Omron CX-Programmer project NewProject (CX-Programmer 9.80)

# PLC NewPLC1: CQM1H CPU51

## Global symbols (name address type ; comment)
0.06 BOOL  ; CAP ZERO ELEV BRAS
0.07 BOOL  ; F-C H ELEV BRAS(active_low)
0.08 BOOL  ; ranger complet
0.09 BOOL  ; F-C H ELEV ROUL
0.11 BOOL  ; F-C SEC ELEV BRAS
0.12 BOOL  ; F-C TIRANT BRAS
100.00 BOOL  ; MONT ELEV BRAS
100.01 BOOL  ; DESCENT ELEV BRAS
100.02 BOOL  ; MONT ELEV ROUL
100.03 BOOL  ; DESCENT ELEV ROUL
100.06 BOOL  ; M-ROUL FIXE
100.10 BOOL  ; VITESSE1 ELEV BRAS
100.11 BOOL  ; VITESSE2 ELEV BRAS
100.13 BOOL  ; VITESSE1 ELEV ROUL
101.00 BOOL  ; VITESSE3 ROUL FIXE
101.08 BOOL  ; FREIN ELEV BRAS
101.09 BOOL  ; FREIN ELEV ROUL
101.10 BOOL  ; INSER COMMANDE
101.11 BOOL  ; SIRENE
101.13 BOOL  ; M-COUROIE ENTREE
102.00 BOOL  ; M-ELEV BRAS
102.01 BOOL  ; M-ROUL BOX
102.02 BOOL  ; OUVER BRAS
102.03 BOOL  ; FERME BRAS
102.06 BOOL  ; SOULEV COURROIE
102.08 BOOL  ; M/D CENTREUR
102.09 BOOL  ; AVANT CHAINE
102.10 BOOL  ; ARRIERE CHAINE
102.11 BOOL  ; VITESSE1 CHAINE
102.12 BOOL  ; PASSARELLA  AVANT
102.14 BOOL  ; PASSARELLA  ARRIERE
102.15 BOOL  ; PASSARELLA  ARRIERE Vitesse 1
116.00 BOOL  ; presence box avec obligation du centrerur ou non box
116.01 BOOL  ; front montant cateur zero elev bras
116.10 BOOL  ; automatique chaine
116.11 BOOL  ; man/auto
117.06 BOOL  ; condition securiter elev rolo en position bas
118.10 BOOL  ; position acutuelle>position de reference
118.11 BOOL  ; position_actuelle<positioin_de_reference
119.14 BOOL  ; button_zero
120.00 BOOL  ; button_zero
120.01 BOOL  ; button_start_cycle_automatique
121.00 BOOL  ; UP_cent_hmi_button
121.01 BOOL  ; descent_centrure_hmi_button
121.02 BOOL  ; BUTTON_chaine_avant_hmi
121.03 BOOL  ; button_chaine_arriere_hmi
140.00 BOOL  ; front mont hr1.00
170.00 BOOL  ; condition monter et frein elev bras
170.01 BOOL  ; condition descente elev bras
1.00 BOOL  ; CAP BRAS OUVERT
1.01 BOOL  ; CAP BRAS FERMEE
1.02 BOOL  ; PH-C DEBORD BOX
1.03 BOOL  ; cap alignement elev rolo et elev bra
1.05 BOOL  ; capteur alignement table fixe et elev rolo
1.06 BOOL  ; CAP COURROIE BAS
1.07 BOOL  ; PH-C FILA CMPL
1.08 BOOL  ; PH-C DEBUT ROUL
1.09 BOOL  ; PH-C STOP FILA
1.10 BOOL  ; PH-C ROUL BOX
1.11 BOOL  ; PH-C P.A.P
1.14 BOOL  ; CENTREUR H
1.15 BOOL  ; CENTREUR BAS
2.00 BOOL  ; COMMANDE INSEREE
2.01 BOOL  ; DCL THERMIQUE
2.02 BOOL  ; ALARME INV
2.04 BOOL  ; switcheur_passarella_arriere
2.05 BOOL  ; switcheur_passarella_avant
2.06 BOOL  ; F-C BOX MACHINE
2.08 BOOL  ; F-C CHAINE AVANT
2.09 BOOL  ; FC_CHAINE_ARRIERE
2.10 BOOL  ; retour_partielle
2.12 BOOL  ; fc_zone_a_passarella
2.13 BOOL  ; passarella_en_avant
2.14 BOOL  ; PASSARELLA_en_arriere
2.15 BOOL  ; fc_zone_b_passarella
70.02 BOOL  ; condition monter elev rolo
70.03 BOOL  ; condition desencete elev rolo
71.03 BOOL  ; COND_Passarella_avnat
71.04 BOOL  ; cond_passarella_arriere
72.06 BOOL  ; condition_centrure
72.08 BOOL  ; condition_centrure
72.09 BOOL  ; condition_chaine_avant
72.10 BOOL  ; condition_chaine_arriere
HR0.00 BOOL  ; start-chargement-box-automatique
HR10.02 BOOL  ; condition pour descent au capteur zero (aligne au box )
HR10.03 BOOL  ; elev bras en  pos 0
HR10.13 BOOL  ; condition 0 elev rouleau
HR10.15 BOOL  ; machine en pos zero
HR11.00 BOOL  ; condition pour start cycle automatique
HR11.01 BOOL  ; condition pour depart du cycle_automatique
HR11.02 BOOL  ; machine en pos initiale avec alignement entre bras et rolo
HR11.03 BOOL  ; condition pour fin du cycle
HR13.00 BOOL  ; chercher table fixe vers l'haut
HR13.01 BOOL  ; chercher table fixe vers le bas
HR13.02 BOOL  ; table mobile  aligne au table fixe
HR13.03 BOOL  ; range complet table fix
HR1.00 BOOL  ; condition pour  elev bra en position exacte et bras fermer
HR1.05 BOOL  ; BT_complet_charging_box
HR2.01 BOOL  ; condition de chercher du elev rolo vers le haut
HR2.02 BOOL  ; condition de chercher du elev bras vers le bas
HR2.03 BOOL  ; condition monter elev rolo en fin du cycle
HR2.04 BOOL  ; condition chercher table fixe  vers le bas
HR2.05 BOOL  ; condition du chercher du table fixe vers le haut
HR3.00 BOOL  ; chaine en automatique
HR3.01 BOOL  ; centrure bas_automatique et manuelle
HR3.02 BOOL  ; etat_box_ready_to_go_out
HR3.03 BOOL  ; etat_BOX_out
HR3.04 BOOL  ; WAIT FOR EMPTY BOX
HR3.05 BOOL  ; BOX IS READY TO ENTER
HR3.06 BOOL  ; condition d'activation cent h man et auto
HR5.04 BOOL  ; Condition alarme generale
HR5.05 BOOL  ; ALARM CENTRURE
HR8.01 BOOL  ; ETAT ARRIERE PASSARELLA

## Program NewProgram1 (no task)

### Section Section1

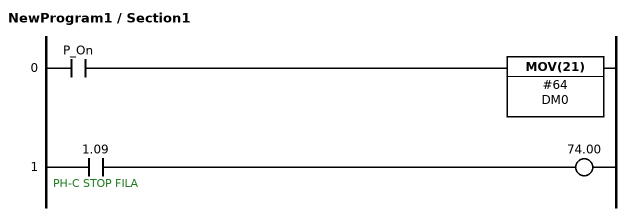
; rung 0
LD P_On
MOV(21) #64 DM0
; rung 1
LD 1.09  ; PH-C STOP FILA
OUT 74.00

### Section Section2

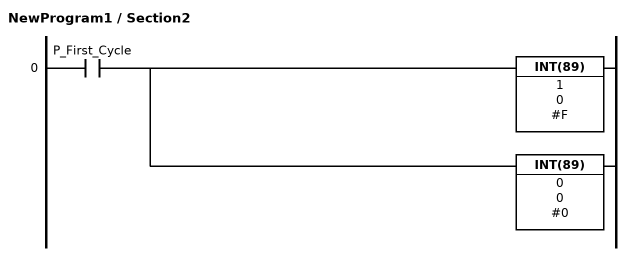
; rung 0
LD P_First_Cycle
INT(89) 1 0 #F
INT(89) 0 0 #0

### Section Section3

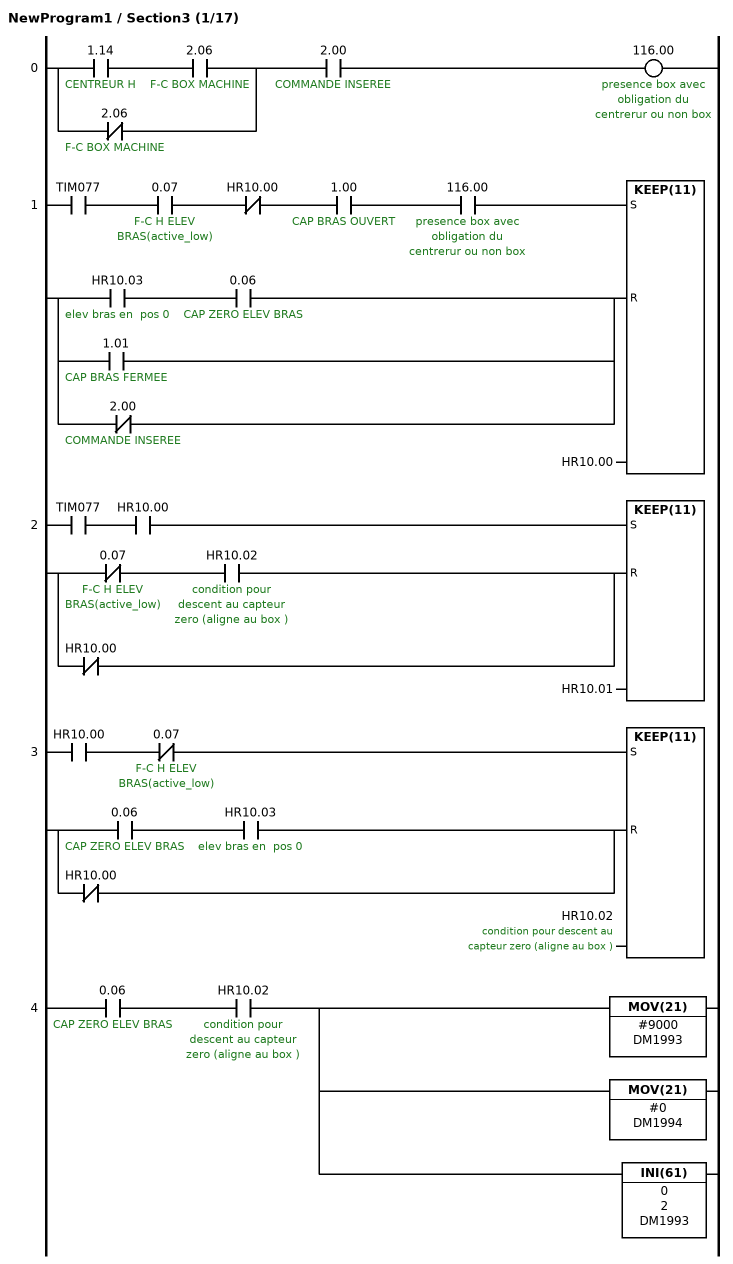
; rung 0
LD 1.14  ; CENTREUR H
AND 2.06  ; F-C BOX MACHINE
ORNOT 2.06  ; F-C BOX MACHINE
AND 2.00  ; COMMANDE INSEREE
OUT 116.00  ; presence box avec obligation du centrerur ou non box
; rung 1
LD TIM077
AND 0.07  ; F-C H ELEV BRAS(active_low)
ANDNOT HR10.00
AND 1.00  ; CAP BRAS OUVERT
AND 116.00  ; presence box avec obligation du centrerur ou non box
LD HR10.03  ; elev bras en  pos 0
AND 0.06  ; CAP ZERO ELEV BRAS
OR 1.01  ; CAP BRAS FERMEE
ORNOT 2.00  ; COMMANDE INSEREE
KEEP(11) HR10.00
; rung 2
LD TIM077
AND HR10.00
LDNOT 0.07  ; F-C H ELEV BRAS(active_low)
AND HR10.02  ; condition pour descent au capteur zero (aligne au box )
ORNOT HR10.00
KEEP(11) HR10.01
; rung 3
LD HR10.00
ANDNOT 0.07  ; F-C H ELEV BRAS(active_low)
LD 0.06  ; CAP ZERO ELEV BRAS
AND HR10.03  ; elev bras en  pos 0
ORNOT HR10.00
KEEP(11) HR10.02  ; condition pour descent au capteur zero (aligne au box )
; rung 4
LD 0.06  ; CAP ZERO ELEV BRAS
AND HR10.02  ; condition pour descent au capteur zero (aligne au box )
MOV(21) #9000 DM1993
MOV(21) #0 DM1994
INI(61) 0 2 DM1993

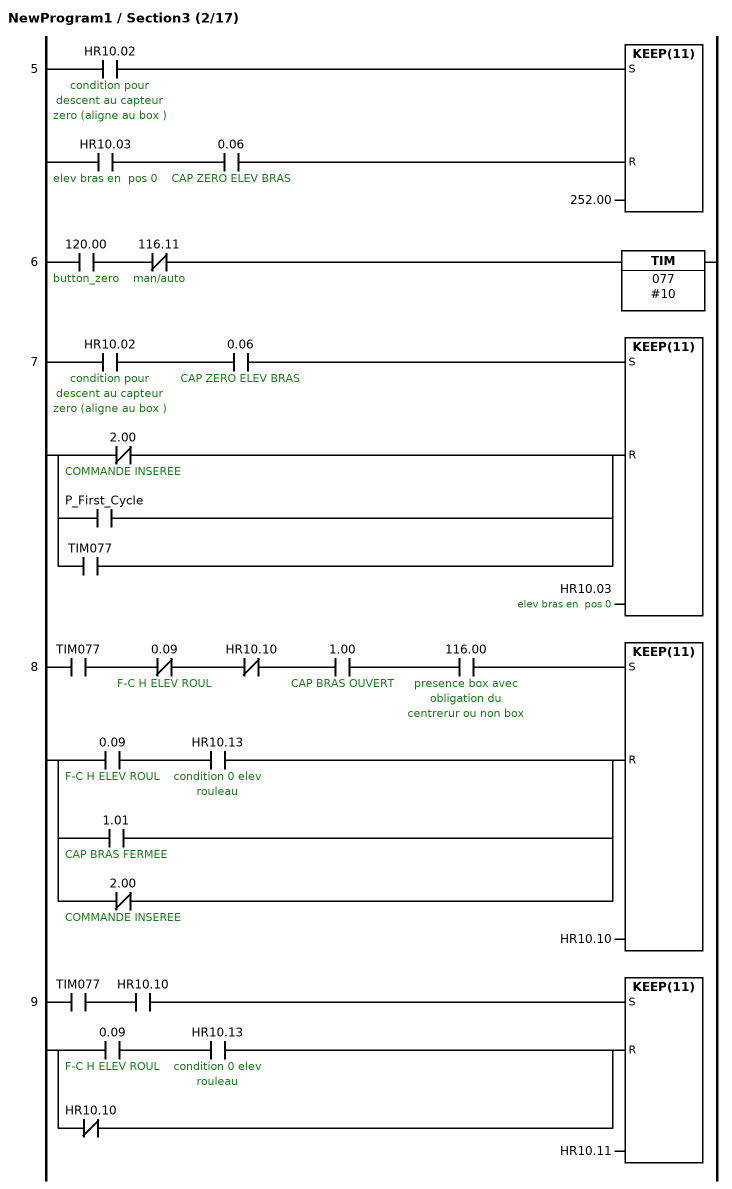
; rung 5
LD HR10.02  ; condition pour descent au capteur zero (aligne au box )
LD HR10.03  ; elev bras en  pos 0
AND 0.06  ; CAP ZERO ELEV BRAS
KEEP(11) 252.00
; rung 6
LD 120.00  ; button_zero
ANDNOT 116.11  ; man/auto
TIM 077 #10
; rung 7
LD HR10.02  ; condition pour descent au capteur zero (aligne au box )
AND 0.06  ; CAP ZERO ELEV BRAS
LDNOT 2.00  ; COMMANDE INSEREE
OR P_First_Cycle
OR TIM077
KEEP(11) HR10.03  ; elev bras en  pos 0
; rung 8
LD TIM077
ANDNOT 0.09  ; F-C H ELEV ROUL
ANDNOT HR10.10
AND 1.00  ; CAP BRAS OUVERT
AND 116.00  ; presence box avec obligation du centrerur ou non box
LD 0.09  ; F-C H ELEV ROUL
AND HR10.13  ; condition 0 elev rouleau
OR 1.01  ; CAP BRAS FERMEE
ORNOT 2.00  ; COMMANDE INSEREE
KEEP(11) HR10.10
; rung 9
LD TIM077
AND HR10.10
LD 0.09  ; F-C H ELEV ROUL
AND HR10.13  ; condition 0 elev rouleau
ORNOT HR10.10
KEEP(11) HR10.11

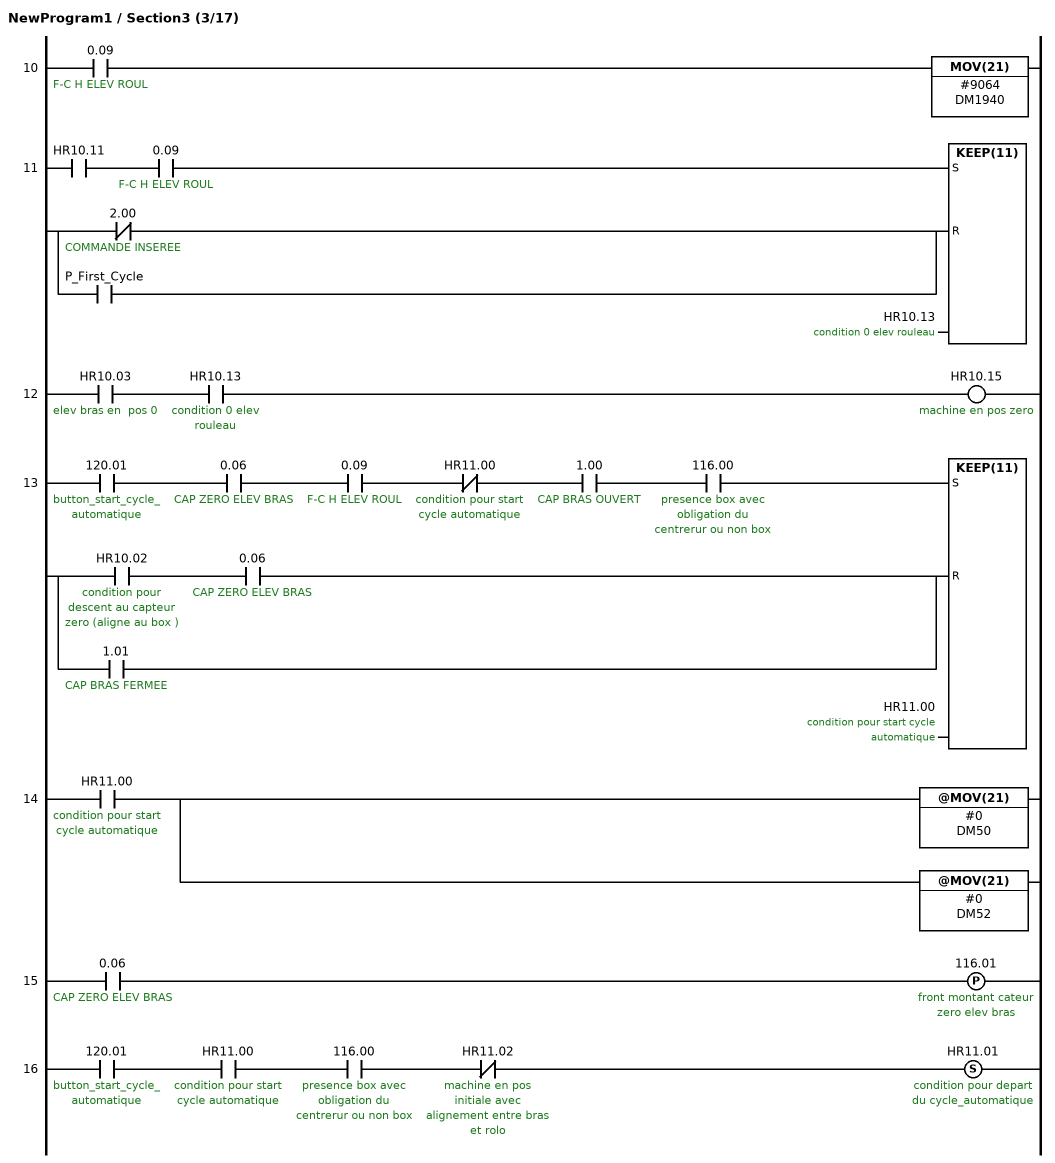
; rung 10
LD 0.09  ; F-C H ELEV ROUL
MOV(21) #9064 DM1940
; rung 11
LD HR10.11
AND 0.09  ; F-C H ELEV ROUL
LDNOT 2.00  ; COMMANDE INSEREE
OR P_First_Cycle
KEEP(11) HR10.13  ; condition 0 elev rouleau
; rung 12
LD HR10.03  ; elev bras en  pos 0
AND HR10.13  ; condition 0 elev rouleau
OUT HR10.15  ; machine en pos zero
; rung 13
LD 120.01  ; button_start_cycle_automatique
AND 0.06  ; CAP ZERO ELEV BRAS
AND 0.09  ; F-C H ELEV ROUL
ANDNOT HR11.00  ; condition pour start cycle automatique
AND 1.00  ; CAP BRAS OUVERT
AND 116.00  ; presence box avec obligation du centrerur ou non box
LD HR10.02  ; condition pour descent au capteur zero (aligne au box )
AND 0.06  ; CAP ZERO ELEV BRAS
OR 1.01  ; CAP BRAS FERMEE
KEEP(11) HR11.00  ; condition pour start cycle automatique
; rung 14
LD HR11.00  ; condition pour start cycle automatique
@MOV(21) #0 DM50
@MOV(21) #0 DM52
; rung 15
LD 0.06  ; CAP ZERO ELEV BRAS
DIFU(13) 116.01  ; front montant cateur zero elev bras
; rung 16
LD 120.01  ; button_start_cycle_automatique
AND HR11.00  ; condition pour start cycle automatique
AND 116.00  ; presence box avec obligation du centrerur ou non box
ANDNOT HR11.02  ; machine en pos initiale avec alignement entre bras et rolo
SET HR11.01  ; condition pour depart du cycle_automatique

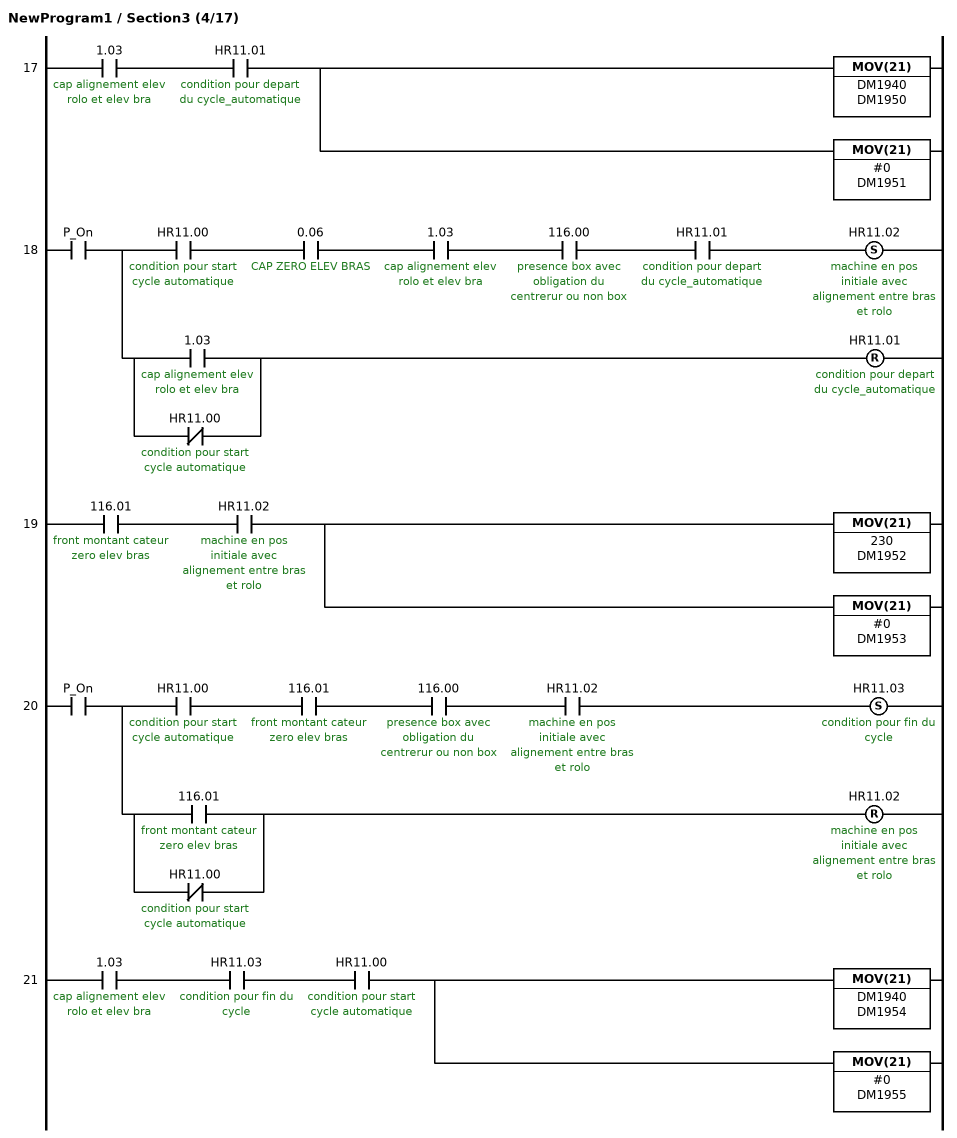
; rung 17
LD 1.03  ; cap alignement elev rolo et elev bra
AND HR11.01  ; condition pour depart du cycle_automatique
MOV(21) DM1940 DM1950
MOV(21) #0 DM1951
; rung 18
LD P_On
OUT TR0
AND HR11.00  ; condition pour start cycle automatique
AND 0.06  ; CAP ZERO ELEV BRAS
AND 1.03  ; cap alignement elev rolo et elev bra
AND 116.00  ; presence box avec obligation du centrerur ou non box
AND HR11.01  ; condition pour depart du cycle_automatique
SET HR11.02  ; machine en pos initiale avec alignement entre bras et rolo
LD TR0
LD 1.03  ; cap alignement elev rolo et elev bra
ORNOT HR11.00  ; condition pour start cycle automatique
ANDLD
RSET HR11.01  ; condition pour depart du cycle_automatique
; rung 19
LD 116.01  ; front montant cateur zero elev bras
AND HR11.02  ; machine en pos initiale avec alignement entre bras et rolo
MOV(21) 230 DM1952
MOV(21) #0 DM1953
; rung 20
LD P_On
OUT TR0
AND HR11.00  ; condition pour start cycle automatique
AND 116.01  ; front montant cateur zero elev bras
AND 116.00  ; presence box avec obligation du centrerur ou non box
AND HR11.02  ; machine en pos initiale avec alignement entre bras et rolo
SET HR11.03  ; condition pour fin du cycle
LD TR0
LD 116.01  ; front montant cateur zero elev bras
ORNOT HR11.00  ; condition pour start cycle automatique
ANDLD
RSET HR11.02  ; machine en pos initiale avec alignement entre bras et rolo
; rung 21
LD 1.03  ; cap alignement elev rolo et elev bra
AND HR11.03  ; condition pour fin du cycle
AND HR11.00  ; condition pour start cycle automatique
MOV(21) DM1940 DM1954
MOV(21) #0 DM1955

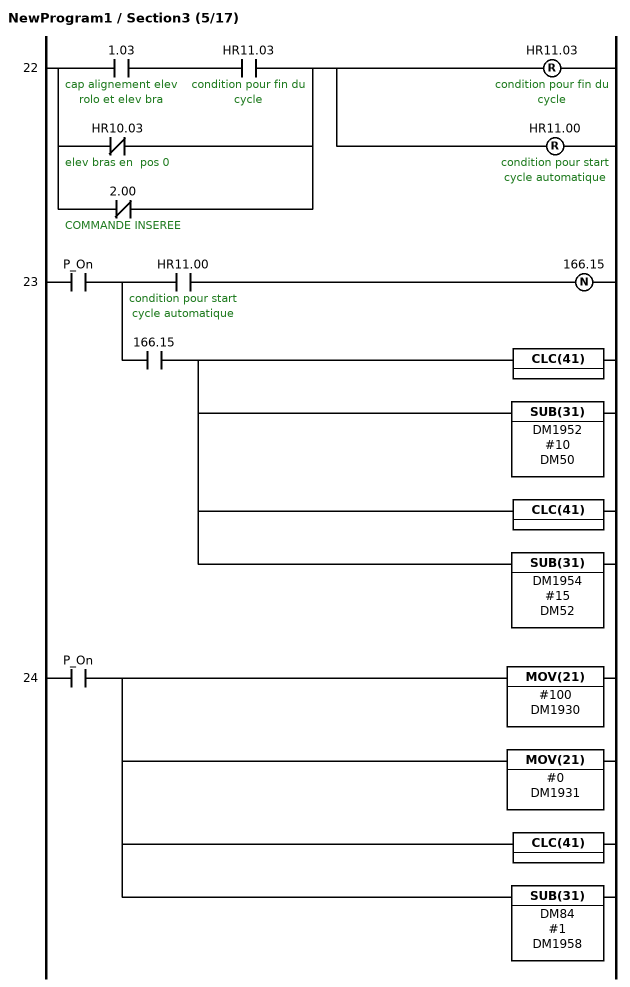
; rung 22
LD 1.03  ; cap alignement elev rolo et elev bra
AND HR11.03  ; condition pour fin du cycle
ORNOT HR10.03  ; elev bras en  pos 0
ORNOT 2.00  ; COMMANDE INSEREE
RSET HR11.03  ; condition pour fin du cycle
RSET HR11.00  ; condition pour start cycle automatique
; rung 23
LD P_On
OUT TR0
AND HR11.00  ; condition pour start cycle automatique
DIFD(14) 166.15
LD TR0
AND 166.15
CLC(41)
SUB(31) DM1952 #10 DM50
CLC(41)
SUB(31) DM1954 #15 DM52
; rung 24
LD P_On
MOV(21) #100 DM1930
MOV(21) #0 DM1931
CLC(41)
SUB(31) DM84 #1 DM1958

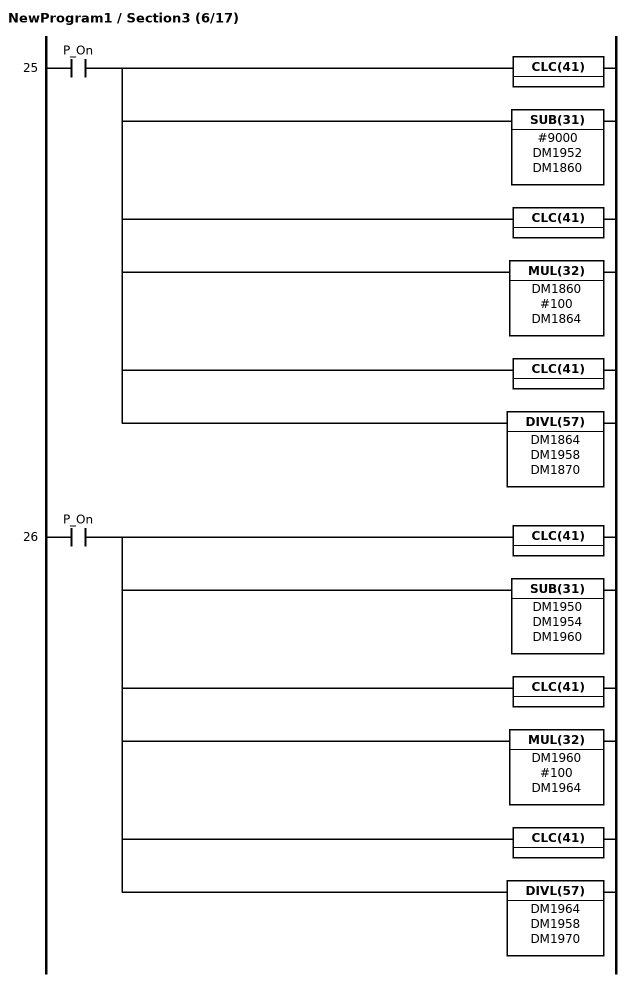
; rung 25
LD P_On
CLC(41)
SUB(31) #9000 DM1952 DM1860
CLC(41)
MUL(32) DM1860 #100 DM1864
CLC(41)
DIVL(57) DM1864 DM1958 DM1870
; rung 26
LD P_On
CLC(41)
SUB(31) DM1950 DM1954 DM1960
CLC(41)
MUL(32) DM1960 #100 DM1964
CLC(41)
DIVL(57) DM1964 DM1958 DM1970

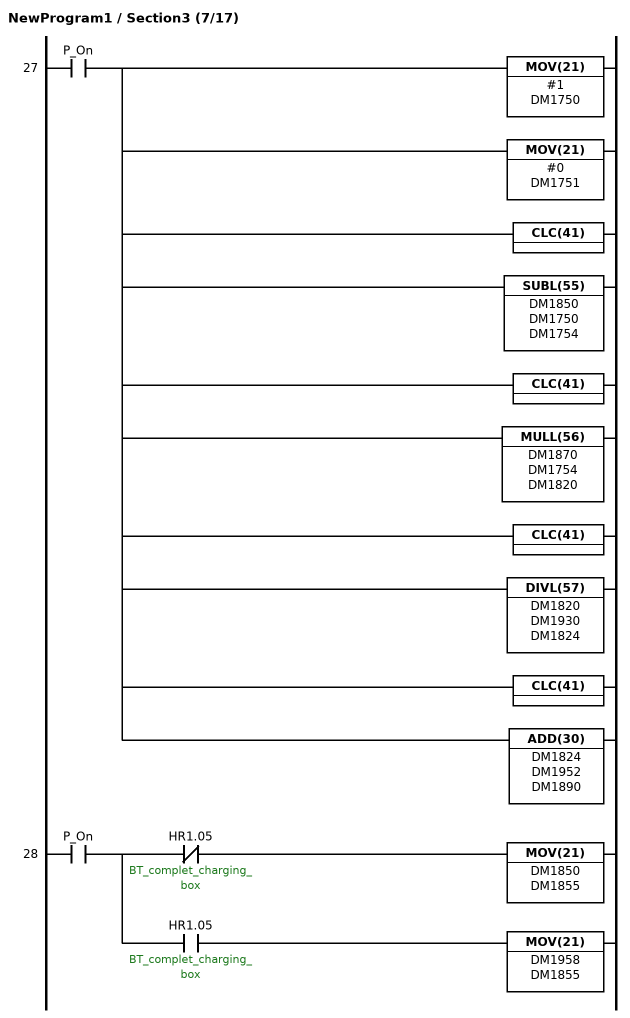
; rung 27
LD P_On
MOV(21) #1 DM1750
MOV(21) #0 DM1751
CLC(41)
SUBL(55) DM1850 DM1750 DM1754
CLC(41)
MULL(56) DM1870 DM1754 DM1820
CLC(41)
DIVL(57) DM1820 DM1930 DM1824
CLC(41)
ADD(30) DM1824 DM1952 DM1890
; rung 28
LD P_On
OUT TR0
ANDNOT HR1.05  ; BT_complet_charging_box
MOV(21) DM1850 DM1855
LD TR0
AND HR1.05  ; BT_complet_charging_box
MOV(21) DM1958 DM1855

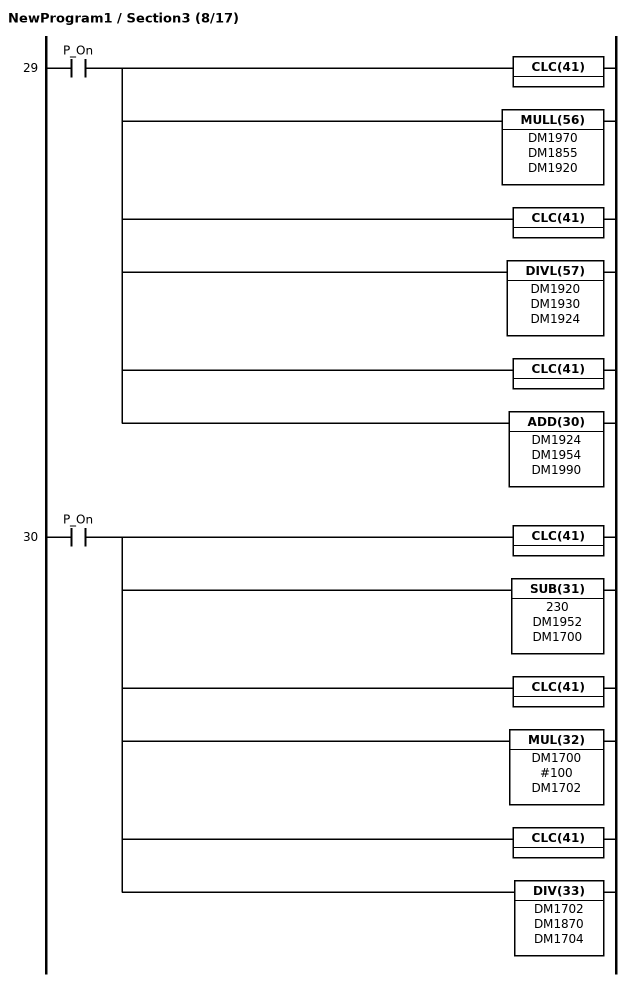
; rung 29
LD P_On
CLC(41)
MULL(56) DM1970 DM1855 DM1920
CLC(41)
DIVL(57) DM1920 DM1930 DM1924
CLC(41)
ADD(30) DM1924 DM1954 DM1990
; rung 30
LD P_On
CLC(41)
SUB(31) 230 DM1952 DM1700
CLC(41)
MUL(32) DM1700 #100 DM1702
CLC(41)
DIV(33) DM1702 DM1870 DM1704

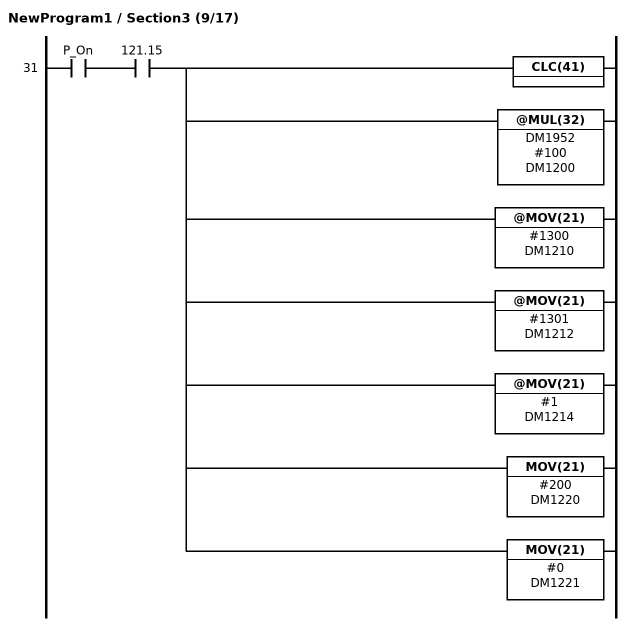
; rung 31
LD P_On
AND 121.15
CLC(41)
@MUL(32) DM1952 #100 DM1200
@MOV(21) #1300 DM1210
@MOV(21) #1301 DM1212
@MOV(21) #1 DM1214
MOV(21) #200 DM1220
MOV(21) #0 DM1221

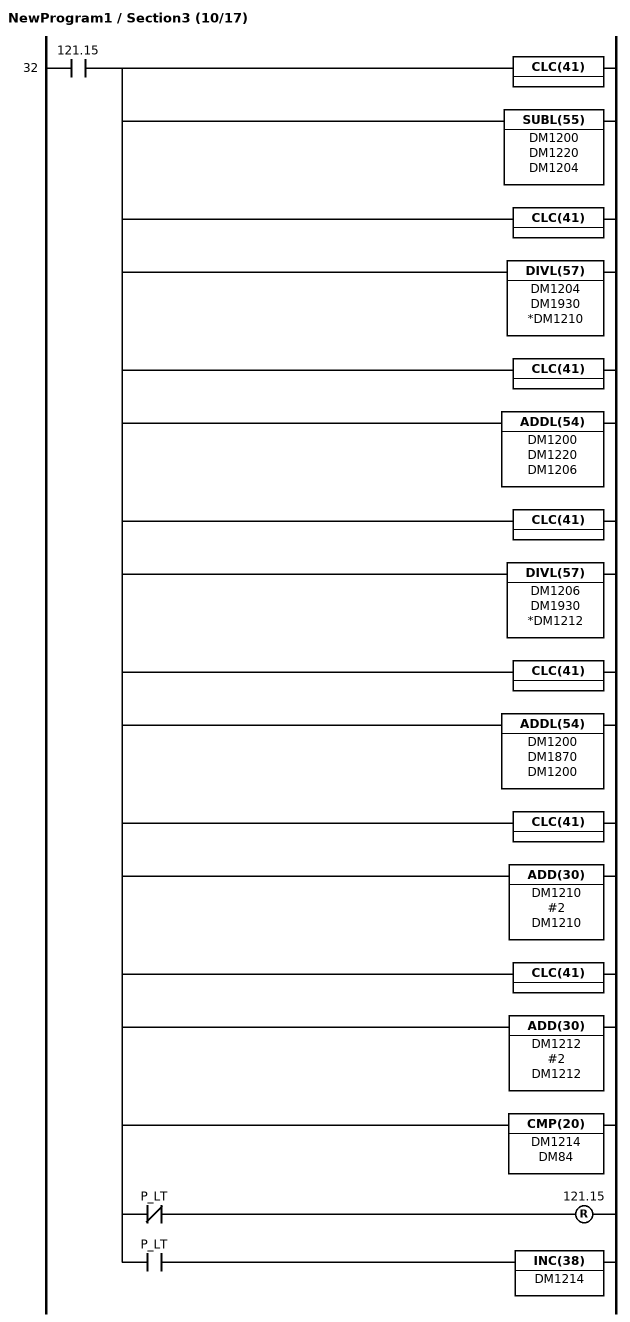
; rung 32
LD 121.15
OUT TR0
CLC(41)
SUBL(55) DM1200 DM1220 DM1204
CLC(41)
DIVL(57) DM1204 DM1930 *DM1210
CLC(41)
ADDL(54) DM1200 DM1220 DM1206
CLC(41)
DIVL(57) DM1206 DM1930 *DM1212
CLC(41)
ADDL(54) DM1200 DM1870 DM1200
CLC(41)
ADD(30) DM1210 #2 DM1210
CLC(41)
ADD(30) DM1212 #2 DM1212
CMP(20) DM1214 DM84
ANDNOT P_LT
RSET 121.15
LD TR0
AND P_LT
INC(38) DM1214

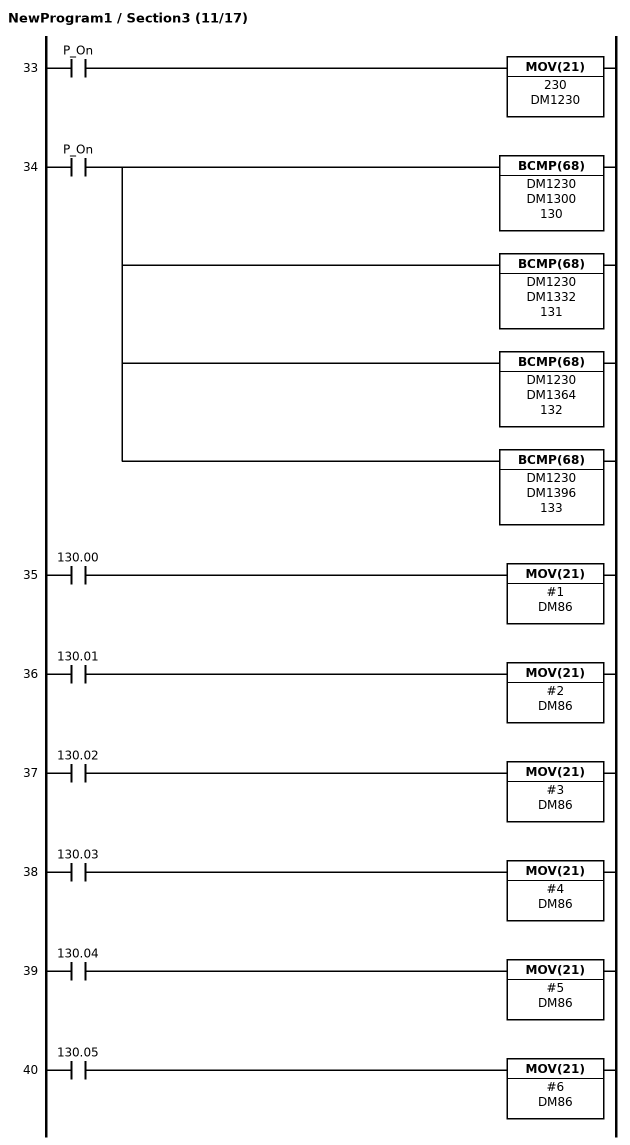
; rung 33
LD P_On
MOV(21) 230 DM1230
; rung 34
LD P_On
BCMP(68) DM1230 DM1300 130
BCMP(68) DM1230 DM1332 131
BCMP(68) DM1230 DM1364 132
BCMP(68) DM1230 DM1396 133
; rung 35
LD 130.00
MOV(21) #1 DM86
; rung 36
LD 130.01
MOV(21) #2 DM86
; rung 37
LD 130.02
MOV(21) #3 DM86
; rung 38
LD 130.03
MOV(21) #4 DM86
; rung 39
LD 130.04
MOV(21) #5 DM86
; rung 40
LD 130.05
MOV(21) #6 DM86

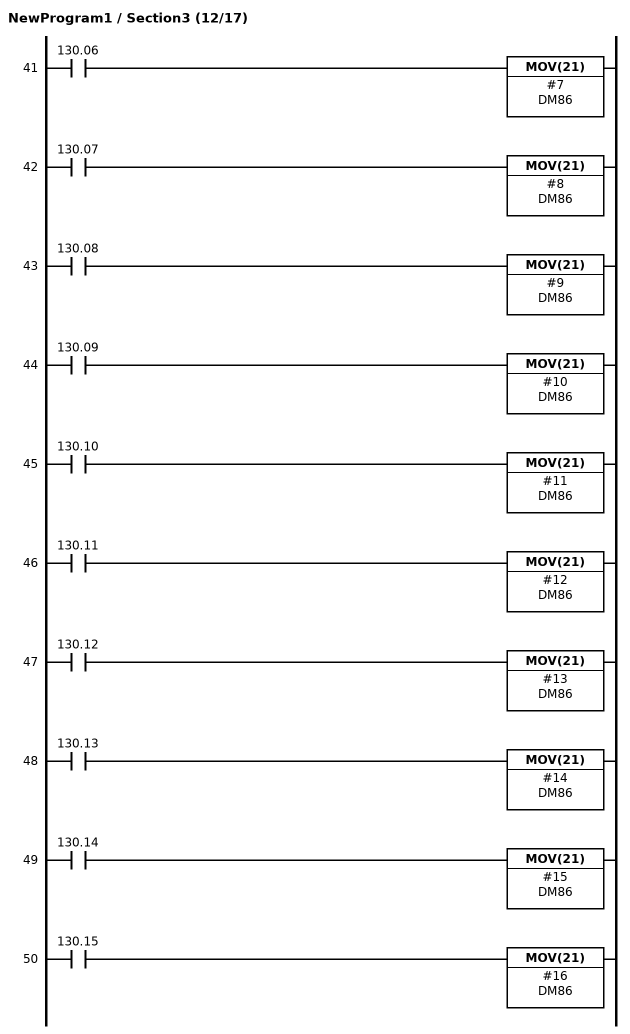
; rung 41
LD 130.06
MOV(21) #7 DM86
; rung 42
LD 130.07
MOV(21) #8 DM86
; rung 43
LD 130.08
MOV(21) #9 DM86
; rung 44
LD 130.09
MOV(21) #10 DM86
; rung 45
LD 130.10
MOV(21) #11 DM86
; rung 46
LD 130.11
MOV(21) #12 DM86
; rung 47
LD 130.12
MOV(21) #13 DM86
; rung 48
LD 130.13
MOV(21) #14 DM86
; rung 49
LD 130.14
MOV(21) #15 DM86
; rung 50
LD 130.15
MOV(21) #16 DM86

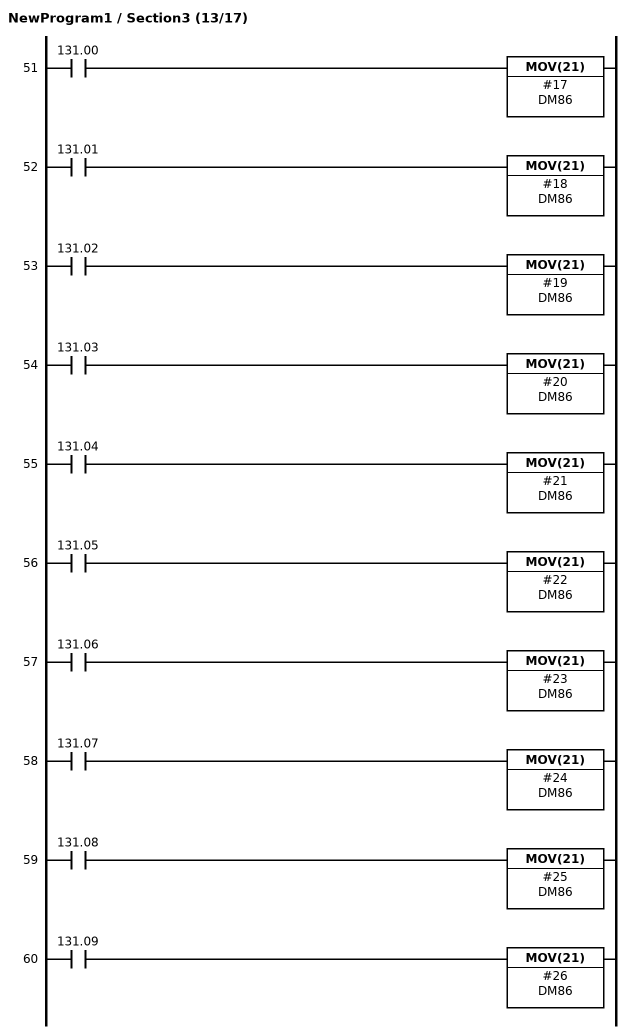
; rung 51
LD 131.00
MOV(21) #17 DM86
; rung 52
LD 131.01
MOV(21) #18 DM86
; rung 53
LD 131.02
MOV(21) #19 DM86
; rung 54
LD 131.03
MOV(21) #20 DM86
; rung 55
LD 131.04
MOV(21) #21 DM86
; rung 56
LD 131.05
MOV(21) #22 DM86
; rung 57
LD 131.06
MOV(21) #23 DM86
; rung 58
LD 131.07
MOV(21) #24 DM86
; rung 59
LD 131.08
MOV(21) #25 DM86
; rung 60
LD 131.09
MOV(21) #26 DM86

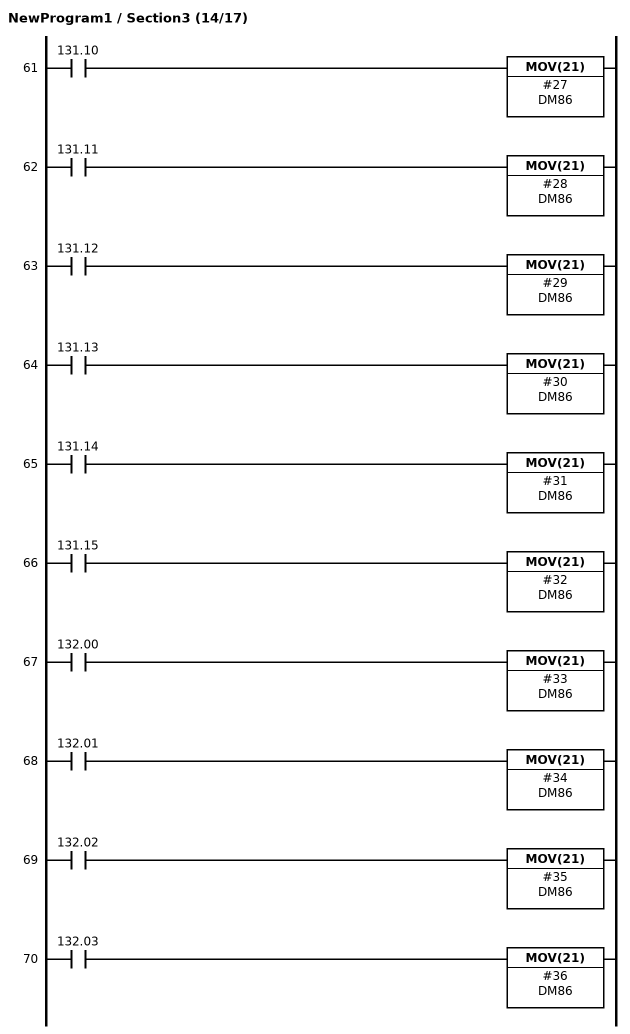
; rung 61
LD 131.10
MOV(21) #27 DM86
; rung 62
LD 131.11
MOV(21) #28 DM86
; rung 63
LD 131.12
MOV(21) #29 DM86
; rung 64
LD 131.13
MOV(21) #30 DM86
; rung 65
LD 131.14
MOV(21) #31 DM86
; rung 66
LD 131.15
MOV(21) #32 DM86
; rung 67
LD 132.00
MOV(21) #33 DM86
; rung 68
LD 132.01
MOV(21) #34 DM86
; rung 69
LD 132.02
MOV(21) #35 DM86
; rung 70
LD 132.03
MOV(21) #36 DM86

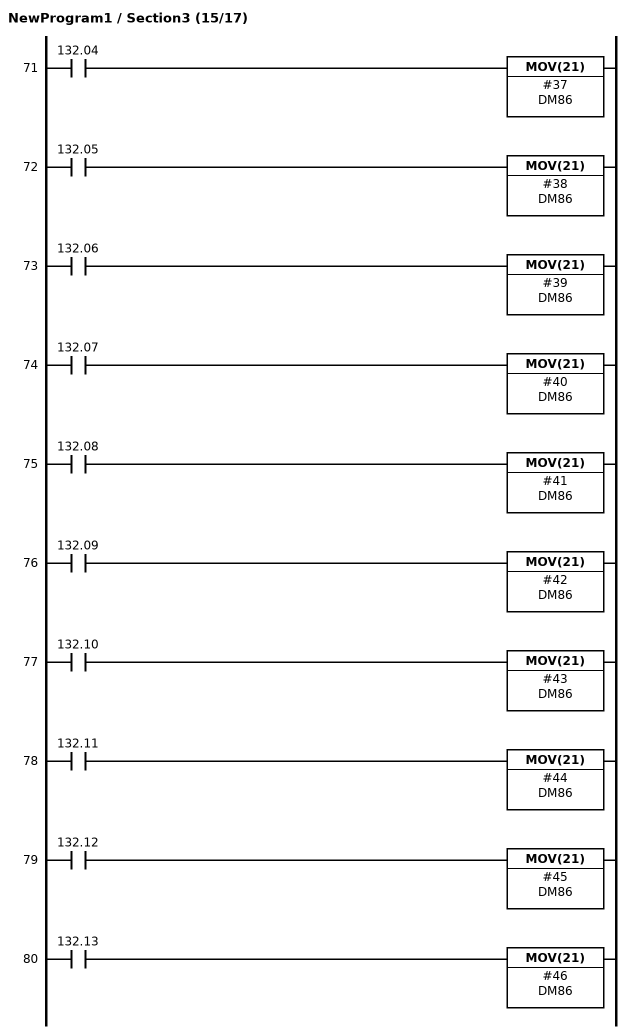
; rung 71
LD 132.04
MOV(21) #37 DM86
; rung 72
LD 132.05
MOV(21) #38 DM86
; rung 73
LD 132.06
MOV(21) #39 DM86
; rung 74
LD 132.07
MOV(21) #40 DM86
; rung 75
LD 132.08
MOV(21) #41 DM86
; rung 76
LD 132.09
MOV(21) #42 DM86
; rung 77
LD 132.10
MOV(21) #43 DM86
; rung 78
LD 132.11
MOV(21) #44 DM86
; rung 79
LD 132.12
MOV(21) #45 DM86
; rung 80
LD 132.13
MOV(21) #46 DM86

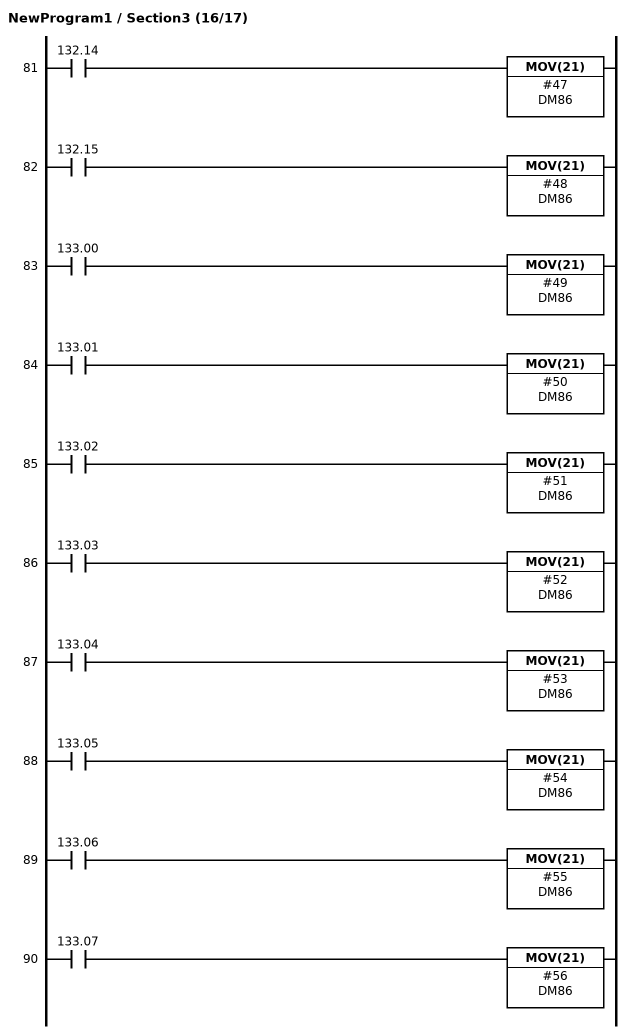
; rung 81
LD 132.14
MOV(21) #47 DM86
; rung 82
LD 132.15
MOV(21) #48 DM86
; rung 83
LD 133.00
MOV(21) #49 DM86
; rung 84
LD 133.01
MOV(21) #50 DM86
; rung 85
LD 133.02
MOV(21) #51 DM86
; rung 86
LD 133.03
MOV(21) #52 DM86
; rung 87
LD 133.04
MOV(21) #53 DM86
; rung 88
LD 133.05
MOV(21) #54 DM86
; rung 89
LD 133.06
MOV(21) #55 DM86
; rung 90
LD 133.07
MOV(21) #56 DM86

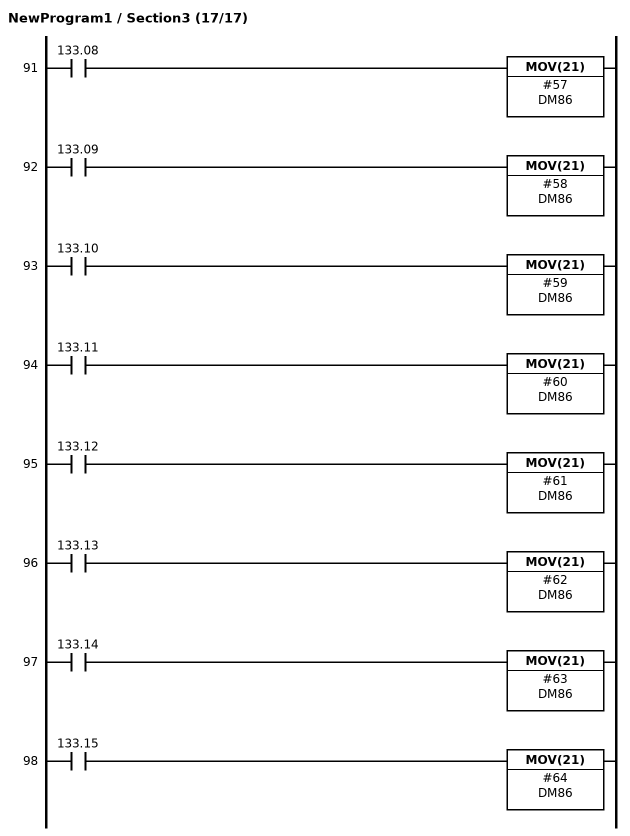
; rung 91
LD 133.08
MOV(21) #57 DM86
; rung 92
LD 133.09
MOV(21) #58 DM86
; rung 93
LD 133.10
MOV(21) #59 DM86
; rung 94
LD 133.11
MOV(21) #60 DM86
; rung 95
LD 133.12
MOV(21) #61 DM86
; rung 96
LD 133.13
MOV(21) #62 DM86
; rung 97
LD 133.14
MOV(21) #63 DM86
; rung 98
LD 133.15
MOV(21) #64 DM86

### Section Section4

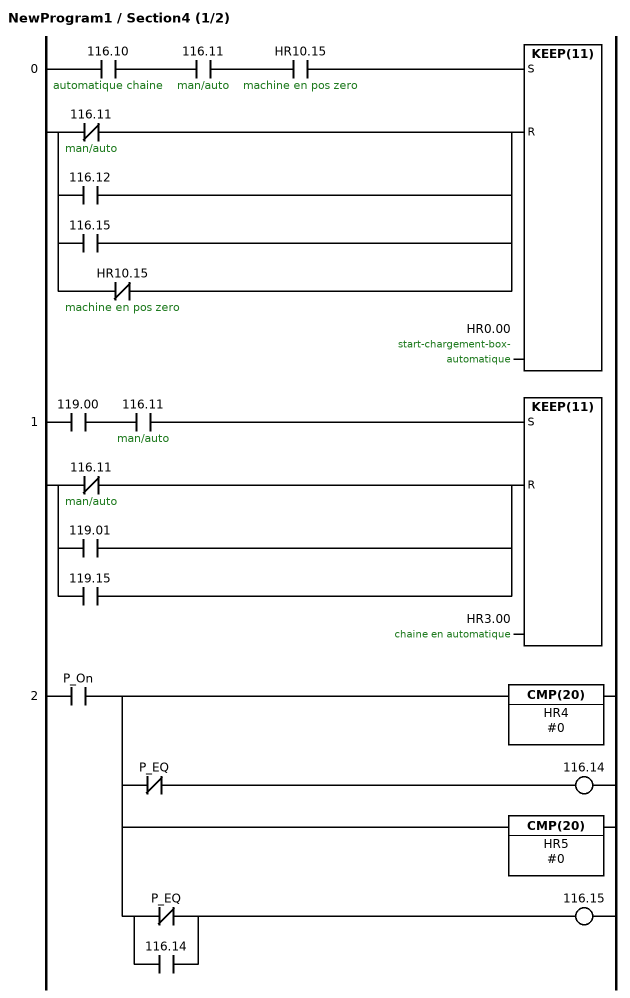
; rung 0
LD 116.10  ; automatique chaine
AND 116.11  ; man/auto
AND HR10.15  ; machine en pos zero
LDNOT 116.11  ; man/auto
OR 116.12
OR 116.15
ORNOT HR10.15  ; machine en pos zero
KEEP(11) HR0.00  ; start-chargement-box-automatique
; rung 1
LD 119.00
AND 116.11  ; man/auto
LDNOT 116.11  ; man/auto
OR 119.01
OR 119.15
KEEP(11) HR3.00  ; chaine en automatique
; rung 2
LD P_On
OUT TR0
CMP(20) HR4 #0
ANDNOT P_EQ
OUT 116.14
LD TR0
CMP(20) HR5 #0
LDNOT P_EQ
OR 116.14
ANDLD
OUT 116.15

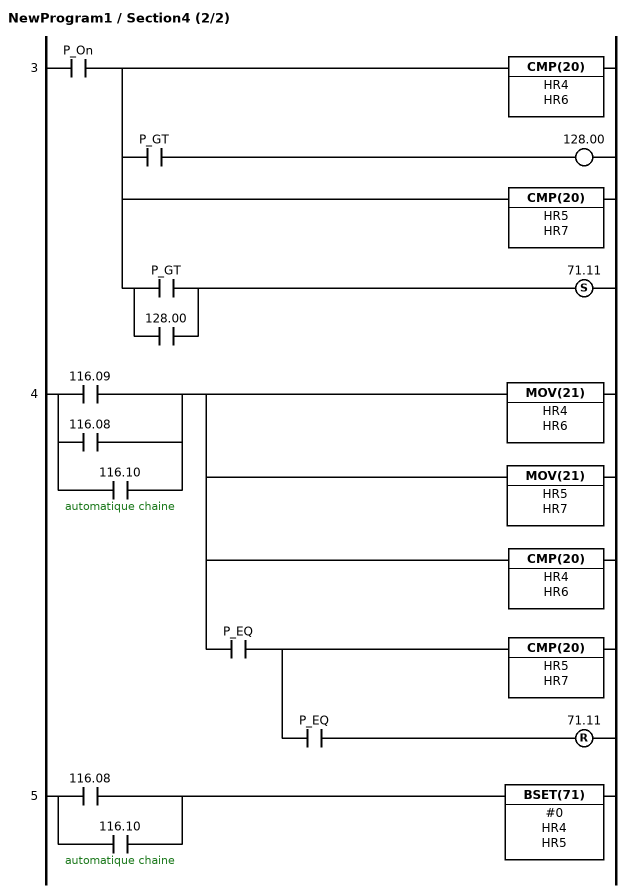
; rung 3
LD P_On
OUT TR0
CMP(20) HR4 HR6
AND P_GT
OUT 128.00
LD TR0
CMP(20) HR5 HR7
LD P_GT
OR 128.00
ANDLD
SET 71.11
; rung 4
LD 116.09
OR 116.08
OR 116.10  ; automatique chaine
MOV(21) HR4 HR6
MOV(21) HR5 HR7
CMP(20) HR4 HR6
AND P_EQ
CMP(20) HR5 HR7
AND P_EQ
RSET 71.11
; rung 5
LD 116.08
OR 116.10  ; automatique chaine
BSET(71) #0 HR4 HR5

### Section Section5

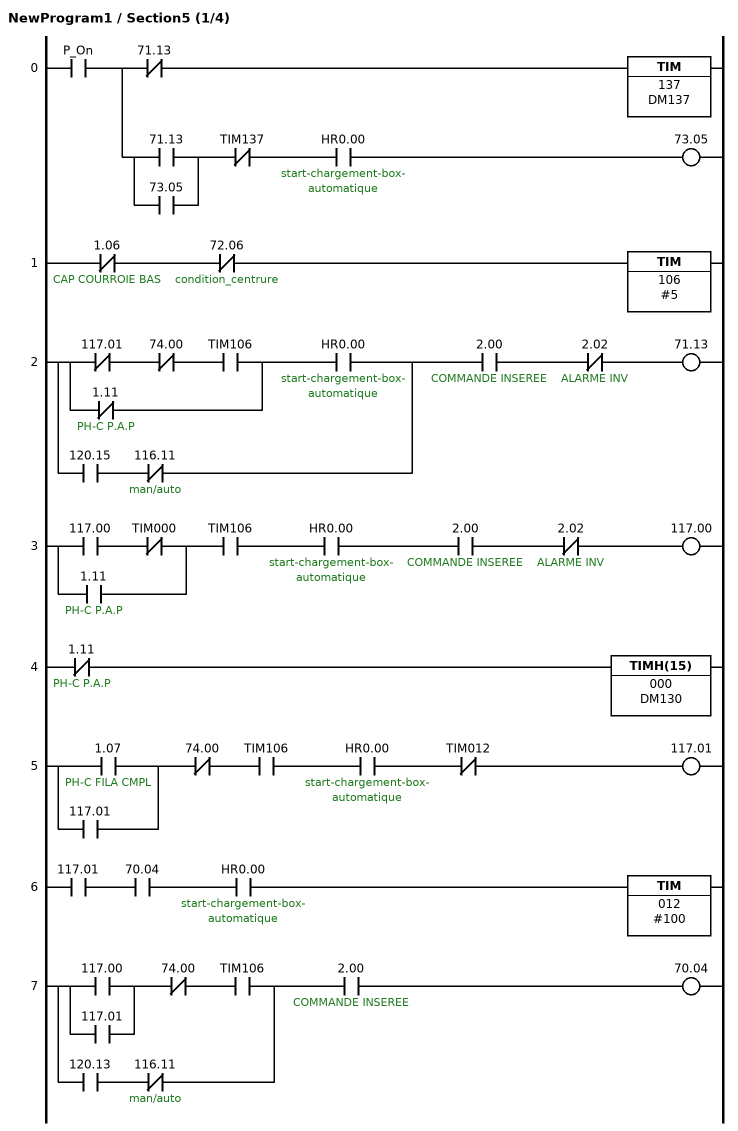
; rung 0
LD P_On
OUT TR0
ANDNOT 71.13
TIM 137 DM137
LD TR0
LD 71.13
OR 73.05
ANDLD
ANDNOT TIM137
AND HR0.00  ; start-chargement-box-automatique
OUT 73.05
; rung 1
LDNOT 1.06  ; CAP COURROIE BAS
ANDNOT 72.06  ; condition_centrure
TIM 106 #5
; rung 2
LDNOT 117.01
ANDNOT 74.00
AND TIM106
ORNOT 1.11  ; PH-C P.A.P
AND HR0.00  ; start-chargement-box-automatique
LD 120.15
ANDNOT 116.11  ; man/auto
ORLD
AND 2.00  ; COMMANDE INSEREE
ANDNOT 2.02  ; ALARME INV
OUT 71.13
; rung 3
LD 117.00
ANDNOT TIM000
OR 1.11  ; PH-C P.A.P
AND TIM106
AND HR0.00  ; start-chargement-box-automatique
AND 2.00  ; COMMANDE INSEREE
ANDNOT 2.02  ; ALARME INV
OUT 117.00
; rung 4
LDNOT 1.11  ; PH-C P.A.P
TIMH(15) 000 DM130
; rung 5
LD 1.07  ; PH-C FILA CMPL
OR 117.01
ANDNOT 74.00
AND TIM106
AND HR0.00  ; start-chargement-box-automatique
ANDNOT TIM012
OUT 117.01
; rung 6
LD 117.01
AND 70.04
AND HR0.00  ; start-chargement-box-automatique
TIM 012 #100
; rung 7
LD 117.00
OR 117.01
ANDNOT 74.00
AND TIM106
LD 120.13
ANDNOT 116.11  ; man/auto
ORLD
AND 2.00  ; COMMANDE INSEREE
OUT 70.04

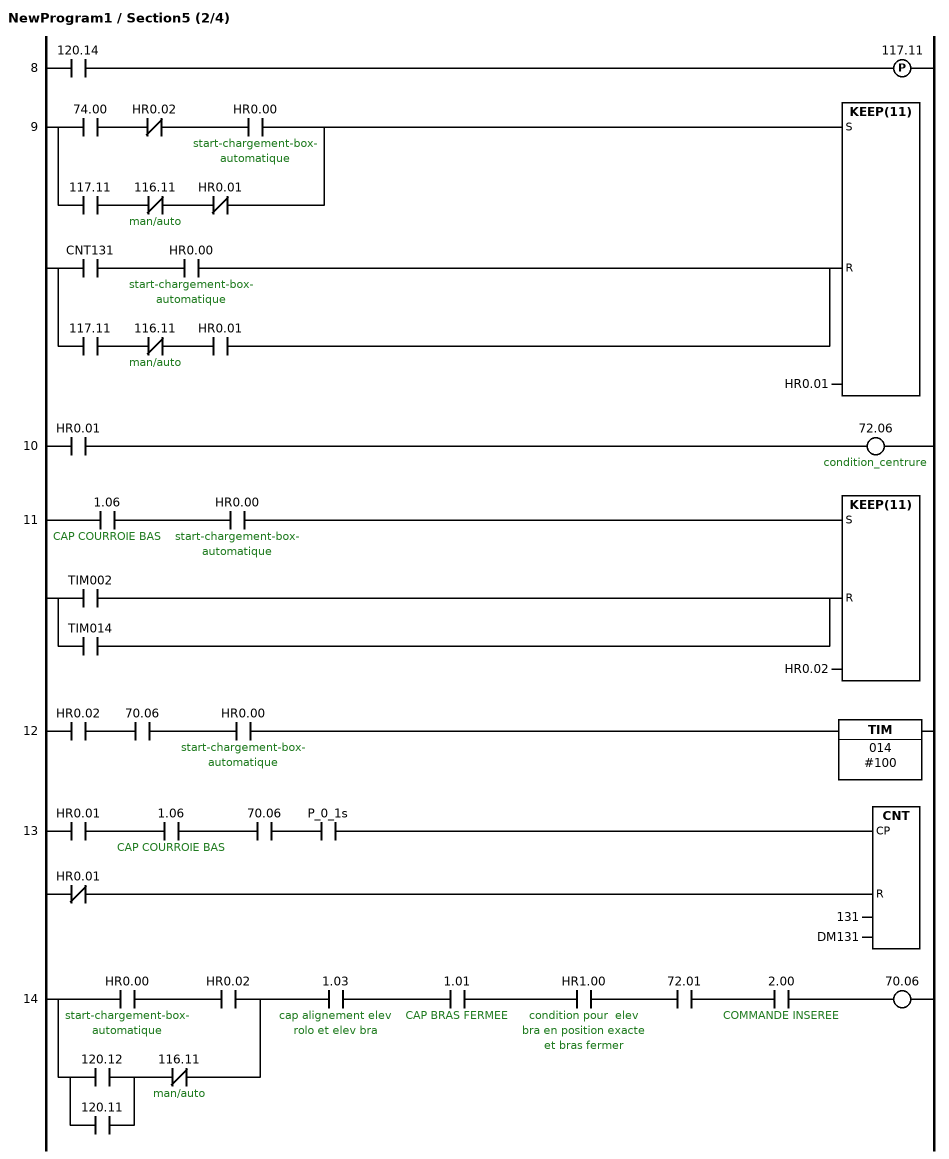
; rung 8
LD 120.14
DIFU(13) 117.11
; rung 9
LD 74.00
ANDNOT HR0.02
AND HR0.00  ; start-chargement-box-automatique
LD 117.11
ANDNOT 116.11  ; man/auto
ANDNOT HR0.01
ORLD
LD CNT131
AND HR0.00  ; start-chargement-box-automatique
LD 117.11
ANDNOT 116.11  ; man/auto
AND HR0.01
ORLD
KEEP(11) HR0.01
; rung 10
LD HR0.01
OUT 72.06  ; condition_centrure
; rung 11
LD 1.06  ; CAP COURROIE BAS
AND HR0.00  ; start-chargement-box-automatique
LD TIM002
OR TIM014
KEEP(11) HR0.02
; rung 12
LD HR0.02
AND 70.06
AND HR0.00  ; start-chargement-box-automatique
TIM 014 #100
; rung 13
LD HR0.01
AND 1.06  ; CAP COURROIE BAS
AND 70.06
AND P_0_1s
LDNOT HR0.01
CNT 131 DM131
; rung 14
LD HR0.00  ; start-chargement-box-automatique
AND HR0.02
LD 120.12
OR 120.11
ANDNOT 116.11  ; man/auto
ORLD
AND 1.03  ; cap alignement elev rolo et elev bra
AND 1.01  ; CAP BRAS FERMEE
AND HR1.00  ; condition pour  elev bra en position exacte et bras fermer
AND 72.01
AND 2.00  ; COMMANDE INSEREE
OUT 70.06

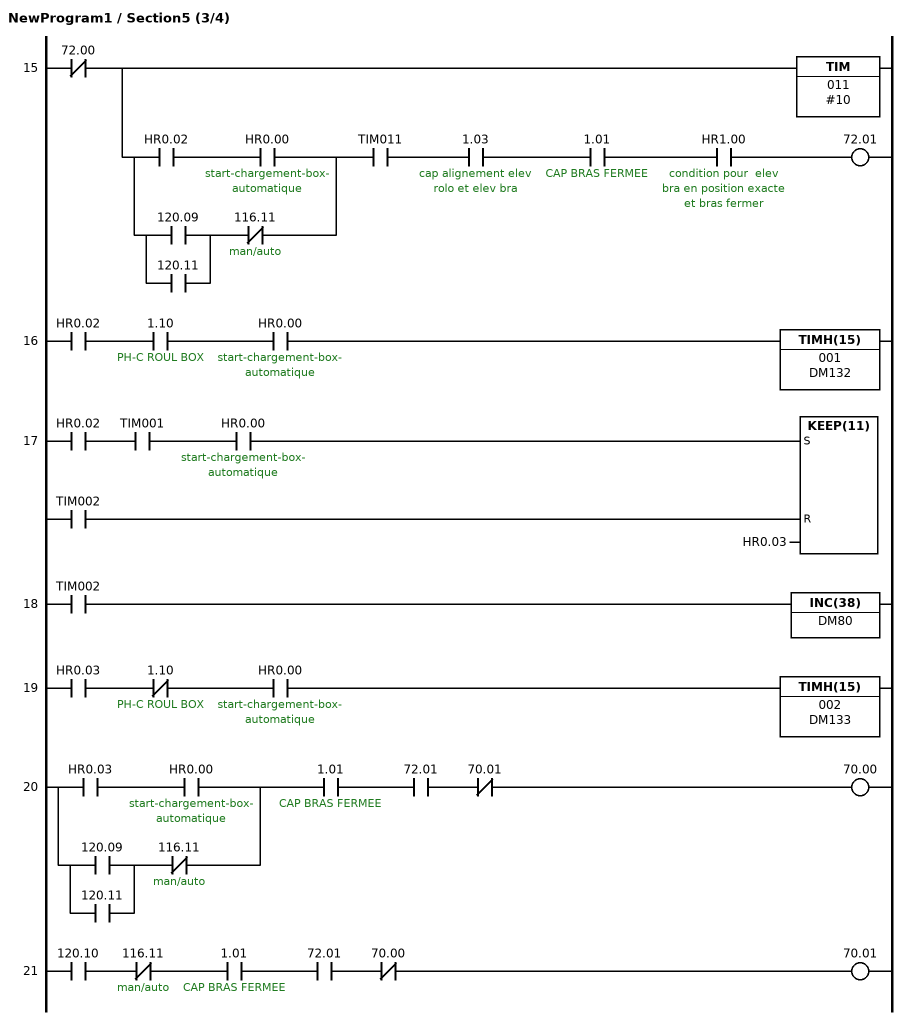
; rung 15
LDNOT 72.00
TIM 011 #10
LD HR0.02
AND HR0.00  ; start-chargement-box-automatique
LD 120.09
OR 120.11
ANDNOT 116.11  ; man/auto
ORLD
ANDLD
AND TIM011
AND 1.03  ; cap alignement elev rolo et elev bra
AND 1.01  ; CAP BRAS FERMEE
AND HR1.00  ; condition pour  elev bra en position exacte et bras fermer
OUT 72.01
; rung 16
LD HR0.02
AND 1.10  ; PH-C ROUL BOX
AND HR0.00  ; start-chargement-box-automatique
TIMH(15) 001 DM132
; rung 17
LD HR0.02
AND TIM001
AND HR0.00  ; start-chargement-box-automatique
LD TIM002
KEEP(11) HR0.03
; rung 18
LD TIM002
INC(38) DM80
; rung 19
LD HR0.03
ANDNOT 1.10  ; PH-C ROUL BOX
AND HR0.00  ; start-chargement-box-automatique
TIMH(15) 002 DM133
; rung 20
LD HR0.03
AND HR0.00  ; start-chargement-box-automatique
LD 120.09
OR 120.11
ANDNOT 116.11  ; man/auto
ORLD
AND 1.01  ; CAP BRAS FERMEE
AND 72.01
ANDNOT 70.01
OUT 70.00
; rung 21
LD 120.10
ANDNOT 116.11  ; man/auto
AND 1.01  ; CAP BRAS FERMEE
AND 72.01
ANDNOT 70.00
OUT 70.01

